// TIA Portal V17 export
// export: Created 2023-05-31T14:08:48.0302768Z, ExportSetting WithDefaults, DisplayName Totally Integrated Automation Portal, DisplayVersion V17, DisplayName TIA Portal Openness, DisplayVersion V17, DisplayName TIA Portal Version Control Interface, DisplayVersion V17, DisplayName STEP 7 Professional, DisplayVersion V17, DisplayName STEP 7 Safety, DisplayVersion V17, DisplayName WinCC Advanced, DisplayVersion V17
FUNCTION_BLOCK "FB_Unit_EDUKIT_PA_Control"   // FB1, LAD
{ S7_Optimized_Access := 'TRUE' }
VERSION : 0.1
// stored: AutoNumber true, IsIECCheckEnabled false, IsRetainMemResEnabled false, MemoryReserve 100, SetENOAutomatically false, UDAEnableTagReadback false
   VAR_INPUT
      Ainput_0 : Int;
      Ainput_1 : Int;
      Ainput_2 : Int;
   END_VAR
   VAR_OUTPUT
      output_startMotor : Bool;
      "output_motorPower [int]" : Int;
      output_valve : Bool;
   END_VAR
   VAR
      startMotor : Bool := true;
      "motorPower [%]" : Real := 85.0;
      valve : Bool;
      "Flow [l/h]" : Real;
      "pressure [mbar]" : Real;
      "pressure [psi]" : Real;
      "level [l]" : Real;
      "step" : Array[0..20] of Bool;
      PID_compact { S7_SetPoint := 'True'} : PID_Compact;
   END_VAR
BEGIN

REGION Network 1
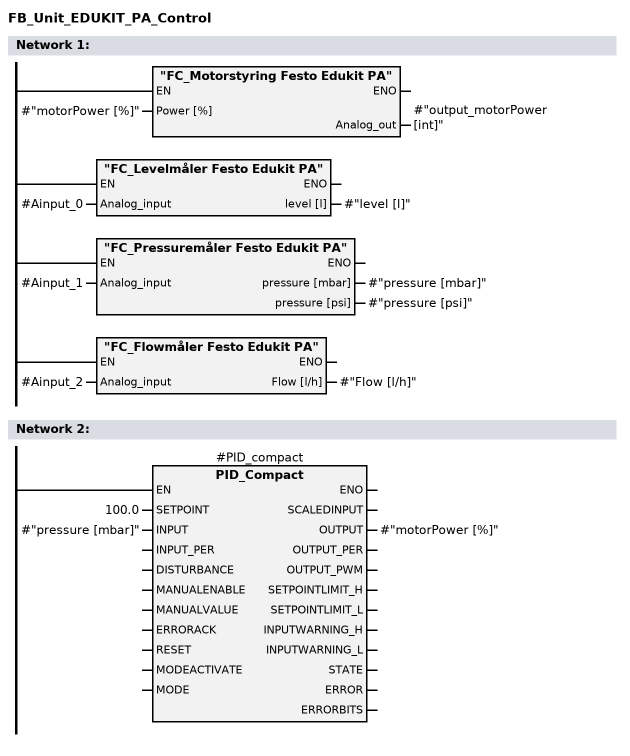
   RUNG wire#powerrail
      "FC_Motorstyring Festo Edukit PA"("Power [%]" := #"motorPower [%]", Analog_out => #"output_motorPower [int]")
   END_RUNG
   RUNG wire#powerrail
      "FC_Levelmåler Festo Edukit PA"(Analog_input := #Ainput_0, "level [l]" => #"level [l]")
   END_RUNG
   RUNG wire#powerrail
      "FC_Pressuremåler Festo Edukit PA"(Analog_input := #Ainput_1, "pressure [mbar]" => #"pressure [mbar]", "pressure [psi]" => #"pressure [psi]")
   END_RUNG
   RUNG wire#powerrail
      "FC_Flowmåler Festo Edukit PA"(Analog_input := #Ainput_2, "Flow [l/h]" => #"Flow [l/h]")
   END_RUNG
   // the same network as SCL:
   "FC_Motorstyring Festo Edukit PA"("Power [%]" := #"motorPower [%]", Analog_out => #"output_motorPower [int]");
   "FC_Levelmåler Festo Edukit PA"(Analog_input := #Ainput_0, "level [l]" => #"level [l]");
   "FC_Pressuremåler Festo Edukit PA"(Analog_input := #Ainput_1,
                           "pressure [mbar]" => #"pressure [mbar]",
                           "pressure [psi]" => #"pressure [psi]");
   "FC_Flowmåler Festo Edukit PA"(Analog_input := #Ainput_2, "Flow [l/h]" => #"Flow [l/h]");
END_REGION

REGION Network 2
   RUNG wire#powerrail
      #PID_compact.PID_Compact(Setpoint := 100.0, Input := #"pressure [mbar]", Input_PER :=, Disturbance :=, ManualEnable :=, ManualValue :=, ErrorAck :=, Reset :=, ModeActivate :=, Mode :=, ScaledInput =>, Output => #"motorPower [%]", Output_PER =>, Output_PWM =>, SetpointLimit_H =>, SetpointLimit_L =>, InputWarning_H =>, InputWarning_L =>, State =>, Error =>, ErrorBits =>)
   END_RUNG
   // the same network as SCL:
   #PID_compact(Setpoint := 100.0, Input := #"pressure [mbar]", Output => #"motorPower [%]");   // PID_Compact
END_REGION

REGION Network 3 (SCL): Output_control
   IF #"output_motorPower [int]" > 30.0 THEN
       #output_startMotor := 1;
   ELSE
       #output_startMotor := 0;
   END_IF;

   #output_valve := 1;
END_REGION
END_FUNCTION_BLOCK
